// TIA Portal project "Mixer" (V16)
// Barrel with mixer, pump, sensors and dosing pumps

(* hardware
DEVICE "S7-1200 station_1"  S7-1200 Station
   slot 0: "Rack_0"  S7-1200 Rack  Rack  V1.0
   slot 1: "PLC_1"  CPU 1215C AC/DC/Rly  6ES7 215-1BG40-0XB0  V4.4
DEVICE "HMI_1"  TP700 Comfort
   slot 0: "HMI_1"  TP700 Comfort  6AV2 124-0GC01-0AX0  16.0.0.0
   slot 1: "HMI_RT_1"  TP700 Comfort  6AV2 124-0GC01-0AX0  16.0.0.0
   slot 5: "HMI_1.IE_CP_1"  PROFINET Interface  16.0.0.0
      slot 1: "PROFINET Interface_1"  PROFINET Interface
         slot 1: "Port_1"  Port
         slot 2: "Port_2"  Port
   slot 7: "HMI_1.MPI/DP_CP_1"  MPI/DP Interface  16.0.0.0
*)

// ===== PLC "PLC_1"  CPU 1215C AC/DC/Rly =====

VAR_GLOBAL   // PLC tag table "DQ"
   "Feed pomp" AT %Q4.0 : Bool;
   "Mixer" AT %Q4.1 : Bool;
   "Emergency Lamp" AT %Q4.2 : Bool;
   "Tag43" AT %Q4.3 : Bool;
   "Tag44" AT %Q4.4 : Bool;
   "Tag45" AT %Q4.5 : Bool;
   "Tag46" AT %Q4.6 : Bool;
   "Tag47" AT %Q4.7 : Bool;
   "Tag48" AT %Q5.0 : Bool;
   "Tag49" AT %Q5.1 : Bool;
   "Tag50" AT %Q5.2 : Bool;
   "Tag51" AT %Q5.3 : Bool;
   "Tag52" AT %Q5.4 : Bool;
END_VAR

VAR_GLOBAL   // PLC tag table "IM"
   "Start feed pomp" AT %M0.0 : Bool;
   "Stop feed pomp" AT %M0.1 : Bool;
   "Emergency stop" AT %M0.2 : Bool;
   "High level" AT %M0.3 : Bool;
   "Low level" AT %M0.4 : Bool;
   "Manhole" AT %M0.5 : Bool;
   "Start feed mixer" AT %M0.6 : Bool;
   "Stop feed mixer" AT %M0.7 : Bool;
   "DI_Run Mixer" AT %M1.0 : Bool;
   "Error Mixer" AT %M1.1 : Bool;
   "State Mixer" AT %MW1 : Int;
   "Run Mixer" AT %M1.3 : Bool;
   "Tag13" AT %M1.4 : Bool;
   "Tag14" AT %M1.5 : Bool;
   "Tag15" AT %M1.6 : Bool;
   "Tag16" AT %M1.7 : Bool;
   "Tag17" AT %M2.0 : Bool;
   "Tag18" AT %M2.1 : Bool;
   "Tag19" AT %M2.2 : Bool;
   "Tag20" AT %M2.3 : Bool;
   "Tag21" AT %M2.4 : Bool;
   "Tag22" AT %M2.5 : Bool;
   "Tag23" AT %M2.6 : Bool;
   "Tag24" AT %M2.7 : Bool;
END_VAR

ORGANIZATION_BLOCK "Main"   // OB1, LAD, ProgramCycle
TITLE = "Main Program Sweep (Cycle)"
{ S7_Optimized_Access := 'TRUE' }
VERSION : 0.1
   VAR_TEMP   // added for the SCL form of the ladder/FBD networks
      _w1 : Bool;
      _w2 : Bool;
   END_VAR
BEGIN

REGION Network 1: Feed pump control
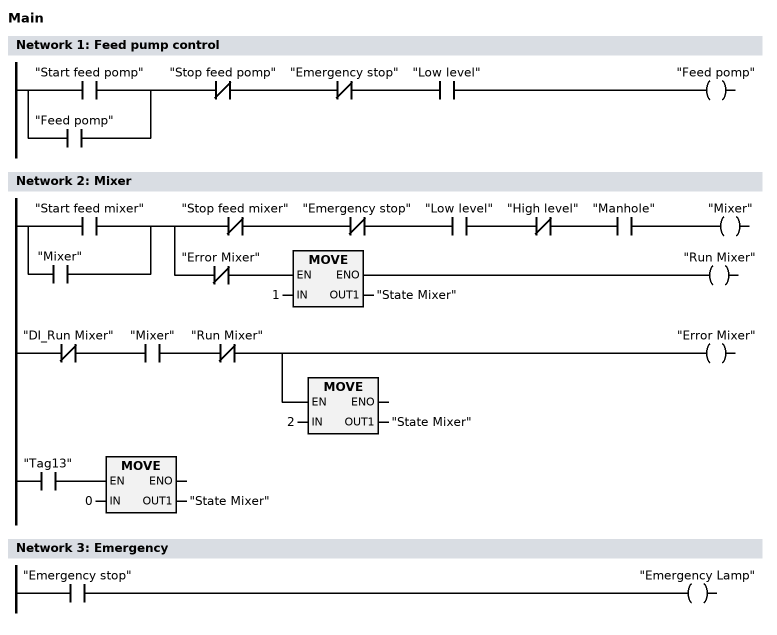
   RUNG wire#powerrail
      Contact( "Start feed pomp" )
      wire#w1
      I_Contact( "Stop feed pomp" )
      I_Contact( "Emergency stop" )
      Contact( "Low level" )
      Coil( "Feed pomp" )
   END_RUNG
   RUNG wire#powerrail
      Contact( "Feed pomp" )
   END_RUNG wire#w1
   // the same network as SCL:
   "Feed pomp" := ("Start feed pomp" OR "Feed pomp") AND NOT "Stop feed pomp" AND NOT "Emergency stop" AND "Low level";
END_REGION

REGION Network 2: Mixer
   RUNG wire#powerrail
      Contact( "Start feed mixer" )
      wire#w1
      I_Contact( "Stop feed mixer" )
      I_Contact( "Emergency stop" )
      Contact( "Low level" )
      I_Contact( "High level" )
      Contact( "Manhole" )
      Coil( "Mixer" )
   END_RUNG
   RUNG wire#powerrail
      Contact( "Mixer" )
   END_RUNG wire#w1
   RUNG wire#w1
      I_Contact( "Error Mixer" )
      Move(in := 1, out1 => "State Mixer")
      Coil( "Run Mixer" )
   END_RUNG
   RUNG wire#powerrail
      I_Contact( "DI_Run Mixer" )
      Contact( "Mixer" )
      I_Contact( "Run Mixer" )
      wire#w2
      Coil( "Error Mixer" )
   END_RUNG
   RUNG wire#w2
      Move(in := 2, out1 => "State Mixer")
   END_RUNG
   RUNG wire#powerrail
      Contact( "Tag13" )
      Move(in := 0, out1 => "State Mixer")
   END_RUNG
   // the same network as SCL:
   #_w1 := "Start feed mixer" OR "Mixer";
   "Mixer" := #_w1 AND NOT "Stop feed mixer" AND NOT "Emergency stop" AND "Low level" AND NOT "High level" AND "Manhole";
   #_w2 := #_w1 AND NOT "Error Mixer";
   IF #_w2 THEN "State Mixer" := 1; END_IF;
   "Run Mixer" := #_w2;
   "Error Mixer" := NOT "DI_Run Mixer" AND "Mixer" AND NOT "Run Mixer";
   IF "Error Mixer" THEN "State Mixer" := 2; END_IF;
   IF "Tag13" THEN "State Mixer" := 0; END_IF;
END_REGION

REGION Network 3: Emergency
   RUNG wire#powerrail
      Contact( "Emergency stop" )
      Coil( "Emergency Lamp" )
   END_RUNG
   // the same network as SCL:
   "Emergency Lamp" := "Emergency stop";
END_REGION
END_ORGANIZATION_BLOCK

(* ===== HMI "HMI_RT_1" =====
system functions are stored by id; their names below are inferred from use
connection "HMI_Connection_1": ETHERNET, S7_1200_OMS

HMI tags "Default tag table"
   "Start feed pomp" : Bool = PLC "Start feed pomp" AT %M0.0, 1 s
   "Start feed mixer" : Bool = PLC "Start feed mixer" AT %M0.6, 1 s
   "Stop feed mixer" : Bool = PLC "Stop feed mixer" AT %M0.7, 1 s
   "Stop feed pomp" : Bool = PLC "Stop feed pomp" AT %M0.1, 1 s
   "Mixer" : Bool = PLC Mixer AT %Q4.1, 1 s
   "Feed pomp" : Bool = PLC "Feed pomp" AT %Q4.0, 1 s
   "Manhole" : Bool = PLC Manhole AT %M0.5, 1 s
   "Low level" : Bool = PLC "Low level" AT %M0.4, 1 s
   "Emergency stop" : Bool = PLC "Emergency stop" AT %M0.2, 1 s
   "State Mixer" : Int = PLC "State Mixer" AT %MW1, 1 s
   "DI_Run Mixer" : Bool = PLC "DI_Run Mixer" AT %M1.0, 1 s

graphic list "Mixer_GR": 0..1 'Graphic_6'; 2..3 'Graphic_5'; 4..5 'Graphic_7'

screen "Home" 800x480
   Button "Button_1" at 13,396 size 134x36; TextOff 'Start'
      on Press: function_b14e0dd5("Start feed mixer", 0)
      Appearance <- "Start feed mixer"
   Button "Button_2" at 13,437 size 134x36; TextOff 'Stop'
      on Press: function_b14e0dd5("Stop feed mixer", 0)
      Appearance <- "Stop feed mixer"
   Button "Button_3" at 151,396 size 134x36; TextOff 'Start'
      Appearance <- "Start feed pomp"
      on Press: function_b14e0dd5("Start feed pomp", 0)
   Button "Button_4" at 151,437 size 134x36; TextOff 'Stop'
      on Press: function_b14e0dd5("Stop feed pomp", 0)
      Appearance <- "Stop feed pomp"
   Circle "Circle_1" at 123,352 size 24x24
      Appearance <- "Mixer"
   Circle "Circle_2" at 255,352 size 24x24
      Appearance <- "Feed pomp"
   Button "Button_5" at 667,13 size 124x32; TextOff 'Two Screen'
      on Press: ActivateScreen("Two Screen", 0)
   TextField "Text field_1" at 20,349 size 84x31; Text 'Mixer'
   TextField "Text field_2" at 163,349 size 84x31; Text 'Pomp'
   Button "Button_6" at 667,56 size 124x32; TextOff 'Demo mode'
      on Press: InvertBit("Manhole"); InvertBit("Low level"); InvertBit("DI_Run Mixer")
      Appearance <- "Manhole"
   Button "Button_7" at 288,396 size 134x36; TextOff 'E - Stop'
      Appearance <- "Emergency stop"
      on Press: SetBit("Emergency stop")
   Button "Button_8" at 288,438 size 134x36; TextOff 'Reset'
      Appearance <- "Emergency stop"
      on Click: ResetBit("Emergency stop")
      on Press: ResetBit("Emergency stop")
   GraphicView "Graphic view_1" at 219,126 size 180x176; Picture "Graphic_4"
      Appearance <- "State Mixer"
   GraphicView "Graphic view_3" at 276,68 size 67x164; Picture "Graphic_6"
   GraphicView "Graphic view_2" at 425,68 size 67x164; Picture "Graphic_5"
   GraphicView "Graphic view_4" at 503,38 size 67x164; Picture "Graphic_7"
   GraphicIOField "Graphic I/O field_1" at 594,90 size 170x110
      ProcessValue <- "State Mixer"

screen "Two Screen" 800x480
   Button "Button_5" at 667,13 size 124x32; TextOff 'Home'
      on Press: ActivateScreen("Home", 0)
*)